{attribute 'qualified_only'}
{attribute 'strict'}
TYPE E_PosDomain :
(
	default := 0,
  master_pos := 1,
//  cycle_pos := 2
  pos_px      := 2     // position in [px]
) UINT;
END_TYPE

(* stored: Version 1.1.0.1, ProductVersion 3.1.4024.3
   EnumerationTextList E_PosDomain: Id {46e45589-f69a-4902-b7ce-94b96f528c23} *)
